// TIA Portal project "flipping mech" (V17)

(* hardware
DEVICE "S7-1500/ET200MP station_1"  S7-1500 station
   slot 0: "Rail_0"  Rack  6ES7 590-1***0-0AA0
   slot 1: "PLC_1"  CPU 1512C-1 PN  6ES7 512-1CK01-0AB0  V2.5
      slot 3: "CPU display_1"  6ES7591-1AA00-0AA0
      slot 32768: "PROFINET interface_1"  X1
         slot 32769: "Port_1"  X1 P1
         slot 32770: "Port_2"  X1 P2
*)

// ===== PLC "PLC_1"  CPU 1512C-1 PN =====

VAR_GLOBAL   // PLC tag table "Default tag table"
   "Tag_1" AT %M0.0 : Bool;
   "Tag_2" AT %M0.1 : Bool;
   "counter" AT %MW100 : Int;
   "i" AT %MW102 : Int;
   "Tag_3" AT %M0.2 : Bool;
END_VAR

DATA_BLOCK "nx"   // DB1
{ S7_Optimized_Access := 'FALSE' }
VERSION : 0.1
   VAR
      gripflip : Int;
      motor : Int;
      linear : Int;
   END_VAR
BEGIN
END_DATA_BLOCK

// folder: System blocks/Program resources

DATA_BLOCK "IEC_Counter_0_DB"   // DB2
{ S7_Optimized_Access := 'TRUE' }
AUTHOR : Simatic
FAMILY : IEC
NAME : CNTR
VERSION : 1.0
// stored: InstanceOfName IEC_COUNTER
"IEC_COUNTER"
BEGIN
END_DATA_BLOCK

DATA_BLOCK "IEC_Timer_0_DB"   // DB3
{ S7_Optimized_Access := 'TRUE' }
AUTHOR : Simatic
FAMILY : IEC
NAME : IEC_TMR
VERSION : 1.0
// stored: InstanceOfName IEC_TIMER
"IEC_TIMER"
BEGIN
END_DATA_BLOCK

DATA_BLOCK "IEC_Timer_0_DB_1"   // DB4
{ S7_Optimized_Access := 'TRUE' }
AUTHOR : Simatic
FAMILY : IEC
NAME : IEC_TMR
VERSION : 1.0
// stored: InstanceOfName IEC_TIMER
"IEC_TIMER"
BEGIN
END_DATA_BLOCK

// folder: (top level)

ORGANIZATION_BLOCK "Main"   // OB1, LAD, ProgramCycle
TITLE = "Main Program Sweep (Cycle)"
{ S7_Optimized_Access := 'TRUE' }
VERSION : 0.1
   VAR_INPUT
      Initial_Call : Bool;   // Initial call of this OB
      Remanence : Bool;   // =True, if remanent data are available
   END_VAR
   VAR_TEMP   // added for the SCL form of the ladder/FBD networks
      _w1 : Bool;
   END_VAR
BEGIN

REGION Network 1
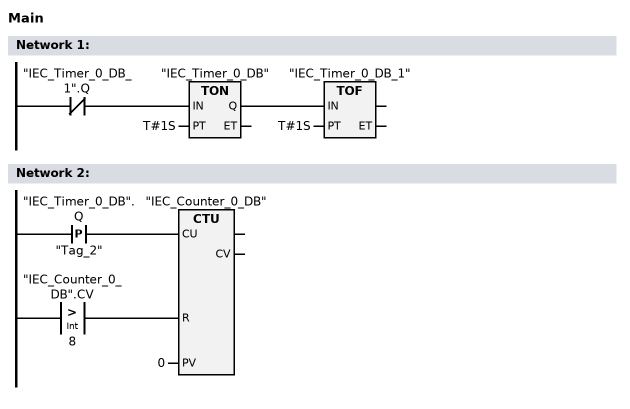
   "IEC_Timer_0_DB".TON(IN := NOT "IEC_Timer_0_DB_1".Q, PT := T#1S);
   "IEC_Timer_0_DB_1".TOF(IN := "IEC_Timer_0_DB".Q, PT := T#1S);
END_REGION

REGION Network 2
   #_w1 := "IEC_Timer_0_DB".Q AND NOT "Tag_2";   // rising edge of "IEC_Timer_0_DB".Q
   "Tag_2" := "IEC_Timer_0_DB".Q;
   "IEC_Counter_0_DB".CTU(CU := #_w1, R := "IEC_Counter_0_DB".CV > 8, PV := 0);
END_REGION

REGION Network 3 (SCL)
   IF "IEC_Counter_0_DB".CV =0 THEN
       "nx".gripflip := 20;
       "nx".linear := 0;
       "nx".motor := 0;
       ;
   END_IF;
   IF "IEC_Counter_0_DB".CV = 1 THEN
       "nx".gripflip := 0;
       "nx".linear := 0;
       "nx".motor := 0;
       ;
   END_IF;
   IF "IEC_Counter_0_DB".CV = 2 THEN
       "nx".gripflip := 0;
       "nx".linear := 80;
       "nx".motor := 0;
       ;
   END_IF;
   IF "IEC_Counter_0_DB".CV = 3 THEN
       "nx".gripflip := 20;
       "nx".linear := 80;
       "nx".motor := 0;
       ;
   END_IF;
   IF "IEC_Counter_0_DB".CV = 4 THEN
       "nx".gripflip := 20;
       "nx".linear := 0;
       "nx".motor := 0;
       ;
   END_IF;
   IF "IEC_Counter_0_DB".CV = 5 THEN
       "nx".gripflip := 20;
       "nx".linear := 0;
       "nx".motor := 180;
       ;
   END_IF;
   IF "IEC_Counter_0_DB".CV = 6 THEN
       "nx".gripflip := 20;
       "nx".linear := 80;
       "nx".motor := 180;
       ;
   END_IF;
   IF "IEC_Counter_0_DB".CV = 7 THEN
       "nx".gripflip := 0;
       "nx".linear := 80;
       "nx".motor := 180;
       ;
   END_IF;
   IF "IEC_Counter_0_DB".CV = 8 THEN
       "nx".gripflip := 0;
       "nx".linear := 0;
       "nx".motor := 180;
       ;
   END_IF;
END_REGION
END_ORGANIZATION_BLOCK